Fanuc TP program (LS listing): _grp_clmp_macro.ls

/PROG  _GRP_CLMP_MACRO	  Macro
/ATTR
OWNER		= MNEDITOR;
COMMENT		= "";
PROG_SIZE	= 203;
CREATE		= DATE 26-06-24  TIME 14:07:08;
MODIFIED	= DATE 26-06-24  TIME 14:07:26;
FILE_NAME	= ;
VERSION		= 0;
LINE_COUNT	= 2;
MEMORY_SIZE	= 567;
PROTECT		= READ_WRITE;
TCD:  STACK_SIZE	= 0,
      TASK_PRIORITY	= 50,
      TIME_SLICE	= 0,
      BUSY_LAMP_OFF	= 0,
      ABORT_REQUEST	= 0,
      PAUSE_REQUEST	= 0;
DEFAULT_GROUP	= *,*,*,*,*;
CONTROL_CODE	= 00000000 00000000;
LOCAL_REGISTERS	= 0,0,0;
/APPL

AUTO_SINGULARITY_HEADER;
  ENABLE_SINGULARITY_AVOIDANCE   : TRUE;
/MN
   1:  DO[65:OFF:Ext Clamp-Up]=(!DO[65:OFF:Ext Clamp-Up]) ;
   2:  DO[66:OFF:Ret Clamp-Down]=(!DO[65:OFF:Ext Clamp-Up]) ;
/POS
/END
